# B&R Automation Studio project AMR_logistics
Automation Studio 6.5.1.7; technology packages: OpcUaCs 6.0.0

## Configuration Config1

CPU 5APC3200.RPL2-000, AutomationRuntime 6.5.1, Build 11.3.0, Vc 6.0.0

### Task classes (Cpu.sw)
```
Cyclic#1:
  PathPlanS1 <- PathPlanST.prg
Cyclic#4:
  RobotAnaly <- RobotAnaly.prg
  MainCtrl <- MainCtrl.prg
```

### Hardware
```
5APC3200_RPL2_000 : 5APC3200.RPL2-000 v1.2.1.0
  Connector IF3:
    AssignedOperatingSystem = ARemb
    ActivateDevice = 1
  Connector IF4:
    AssignedOperatingSystem = ARemb
    ActivateDevice = 1
  Connector IF5:
    AssignedOperatingSystem = ARemb
  Connector IF6:
    AssignedOperatingSystem = ARemb
  Connector IF7:
    AssignedOperatingSystem = ARemb
  Connector IF8:
    AssignedOperatingSystem = ARemb
  ConfigurationID = AMR_logistics_Config1
  Simulation = 1
  FileDevice1
  FileDeviceName1 = USER
  FileDevicePath1 = USER_PATH
```

## Logical view

### Global.var - Global variables
```iecst
VAR_GLOBAL
	gRobotState    : USINT := 0;       (* 0= Idle, 1= Active, 2= Fault *)
	gPosY          : REAL  := 0.0;     (* Robot Y coordinate in meters *)
	gPosX          : REAL  := 0.0;     (* Robot X coordinate in meters *)
	gEmergencyStop : BOOL  := FALSE;   (* E-Stop Signal *)
	gBatteryLevel  : REAL  := 100.0;   (* Battery % - Starts full *)
	gRobotReady    : BOOL  := FALSE;   (* Set by MainControl LD *)
END_VAR
```

### Program Logical/PathPlanST (IEC)

#### Variables.var
```iecst
VAR
	L_VelocityX  : REAL  := 0.05;
	L_VelocityY  : REAL  := 0.02;
	L_StepCount  : UDINT := 0;
END_VAR
```

#### Main.st
```iecst
PROGRAM _CYCLIC

	IF gRobotReady AND (gRobotState = 1) THEN
		gPosX := gPosX + L_VelocityX;
		gPosY := gPosY + L_VelocityY;
		L_StepCount := L_StepCount + 1;
		IF gPosX > 100.0 THEN gPosX := 0.0; END_IF;
		IF gPosY > 100.0 THEN gPosY := 0.0; END_IF;
	END_IF;

END_PROGRAM
```

### Program Logical/RobotAnaly (IEC)

#### Variables.var
```iecst
VAR
	L_DrainRate  : REAL := 0.005;
	L_LowBattWrn : BOOL := FALSE;
	L_CritLevel  : REAL := 10.0;
END_VAR
```

#### Main.st
```iecst
PROGRAM _CYCLIC

	IF gRobotState = 1 THEN
		gBatteryLevel := gBatteryLevel - L_DrainRate;
	END_IF;

	IF gBatteryLevel < 0.0 THEN
		gBatteryLevel := 0.0;
		gRobotState   := 2;
	END_IF;

	IF gBatteryLevel < L_CritLevel THEN
		L_LowBattWrn := TRUE;
	END_IF;

END_PROGRAM
```

### Program Logical/MainCtrl (IEC)

#### Cyclic.ld
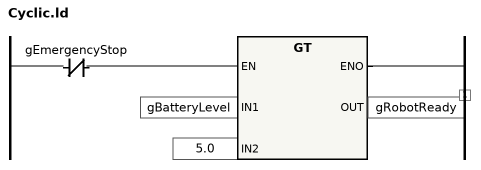
Diagram, in the editor's own instruction-list form stored in the file:
```il
PROGRAM _CYCLIC

VAR
	zz$$$$_0_Eno_GT : BOOL;
END_VAR

{NetworkNumber := 1}
LDN	gEmergencyStop
ST	zz$$$$_0_Eno_GT
LD	zz$$$$_0_Eno_GT
JMPCN ll$$$$_IF_0
LD	gBatteryLevel
GT	5.0
ST	gRobotReady
ll$$$$_IF_0:

END_PROGRAM
```

Listed in the project but not available here: Logical/Global.typ, Logical/Libraries
